PROGRAM P_Task2
VAR
END_VAR

END_PROGRAM

(* stored: Version 1.1.0.1, ProductVersion 3.1.4024.12
   POU P_Task2: Id {ea31129f-1a01-4c4f-861c-0e066cae28a0}, SpecialFunc None *)
